// TIA Portal V17 export
// export: Created 2023-04-04T13:27:27.0343927Z, ExportSetting WithDefaults, DisplayName Totally Integrated Automation Portal, DisplayVersion V17, DisplayName TIA Portal Openness, DisplayVersion V17, DisplayName TIA Portal Version Control Interface, DisplayVersion V17, DisplayName STEP 7 Professional, DisplayVersion V17, DisplayName STEP 7 Safety, DisplayVersion V17, DisplayName WinCC Advanced, DisplayVersion V17
DATA_BLOCK "PRG_VGR_Axis_vertical_Act_Pos_DB"   // DB29
AUTHOR : A.Schaefer
VERSION : 0.1
// stored: AutoNumber true, DBAccessibleFromOPCUA true, DBAccessibleFromWebserver true, InstanceOfName PRG_VGR_Axis_vertical_Act_Pos, InstanceOfType FB
"PRG_VGR_Axis_vertical_Act_Pos"
   // VAR
   //    lfb_IN_DEC { ExternalAccessible := 'False'; ExternalVisible := 'False'; ExternalWritable := 'False'} : "FB_INC_DEC";
   // END_VAR
BEGIN
END_DATA_BLOCK
